Universal Robots PolyScope program: Hospital_big_top.urp

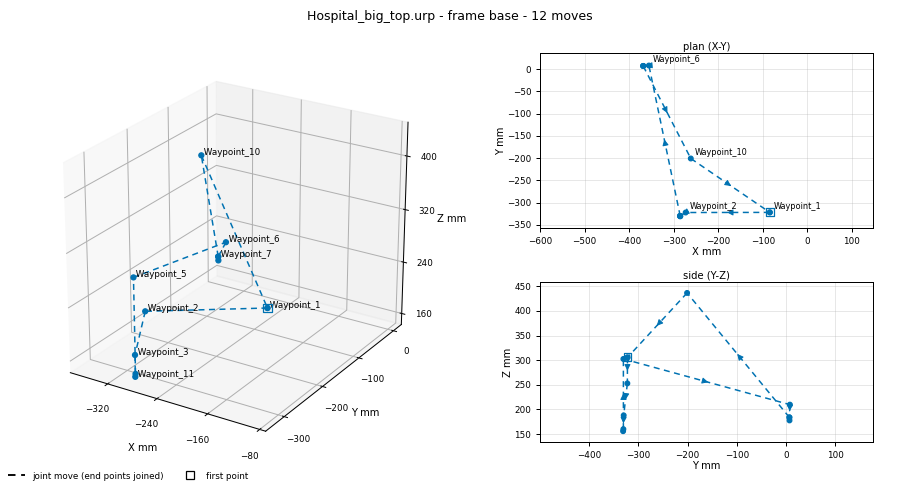
[picture p0: tool path of Hospital_big_top.urp in frame base, 12 of 12 moves have a stored position in this frame; points joined in program order, loops and branches not executed]
Program Hospital_big_top (installation=default directory=/programs/usbdisk/Zahra1 createdIn=5.11.11.1010533 lastSavedIn=5.11.11.1010533 robotSerialNumber=20205300864)
Calibrated DH parameters: a=[-0.000166, -0.243494, -0.153108, 0.000057, -0.000123, 0]; d=[0.151897, -1.34267, 53.988124, -52.514559, 0.085283, 0.092193]; alpha=[1.572472, -0.003756, 0.002824, 1.570807, -1.572621, 0]; deltaTheta=[0, 0.020704, 7.033215, -0.770746, 0.000004, 0]
Robot Program (runOnlyOnce=true)
  MoveJ speed 60 deg/s, acceleration 80 deg/s^2 (useActiveTCP=true) feature=Base
    Waypoint Waypoint_1: TCP in base x=-84.301 y=-321.874 z=305.493 mm, rx=-2.081 ry=-2.2572 rz=0.0985 rad; joints [-79.979, -91.199, -87.973, -91.694, 84.673, 815.506] deg
    URCap Gripper (Robotiq_Grippers, Robotiq Inc.) dataModel(position=46.666666666666664, force=70.0, speed=27.0, positionInDouble=46.666666666666664, forceInDouble=70.0, speedInDouble=27.0, slaveIds=[9], blocking=true, robotCompliant=false)
    Waypoint Waypoint_2: TCP in base x=-273.269 y=-322.149 z=252.836 mm, rx=-2.1606 ry=-2.2563 rz=0.1197 rad; joints [-111.769, -113.952, -75.591, -76.612, 87.489, 785.766] deg
    Waypoint Waypoint_3: TCP in base x=-286.068 y=-329.572 z=187.877 mm, rx=-2.1263 ry=-2.267 rz=0.0386 rad; joints [-113.094, -122.394, -79.226, -67.597, 87.665, 783.343] deg
    Waypoint Waypoint_11: TCP in base x=-285.496 y=-330.769 z=155.775 mm, rx=-2.2131 ry=-2.1958 rz=0.033 rad; joints [-113.09, -125.834, -82.835, -60.62, 88.212, 787.48] deg
    URCap Gripper (Robotiq_Grippers, Robotiq Inc.) dataModel(position=83.92156862745098, force=70.0, speed=27.0, positionInDouble=83.92156862745098, forceInDouble=70.0, speedInDouble=27.0, slaveIds=[9], blocking=true, robotCompliant=true)
    Waypoint Waypoint_4: motionParameters(jointSpeed=0.698132 jointAcceleration=0.523599 cartesianSpeed=0.25 cartesianAcceleration=1.2); TCP in base x=-285.424 y=-330.196 z=159.912 mm, rx=-2.2127 ry=-2.1963 rz=0.0331 rad; joints [-113.112, -125.264, -82.578, -61.439, 88.221, 787.435] deg
    Waypoint Waypoint_5: TCP in base x=-285.408 y=-330.203 z=302.436 mm, rx=-2.2127 ry=-2.1963 rz=0.0332 rad; joints [-113.041, -118.934, -53.354, -96.993, 88.181, 787.434] deg
    Waypoint Waypoint_6: TCP in base x=-355.712 y=7.819 z=209.704 mm, rx=-3.108 ry=-0.037 rz=0.0524 rad; joints [-159.113, -101.607, -103.522, -63.61, 87.579, 829.653] deg
    Waypoint Waypoint_7: TCP in base x=-368.599 y=6.796 z=183.845 mm, rx=-3.106 ry=0.0502 rz=-0.025 rad; joints [-159.969, -108.043, -101.533, -61.904, 88.456, 832.067] deg
    Waypoint Waypoint_8: motionParameters(jointSpeed=0.523599 jointAcceleration=0.349066 cartesianSpeed=0.25 cartesianAcceleration=1.2); TCP in base x=-368.491 y=7.024 z=177.653 mm, rx=-3.106 ry=0.0502 rz=-0.025 rad; joints [-160.001, -108.773, -102.426, -60.281, 88.455, 832.04] deg
    URCap Gripper (Robotiq_Grippers, Robotiq Inc.) dataModel(position=52.549019607843135, force=70.0, speed=18.0, positionInDouble=52.549019607843135, forceInDouble=70.0, speedInDouble=18.0, slaveIds=[9], blocking=true, robotCompliant=true)
    Waypoint Waypoint_7: TCP in base x=-368.599 y=6.796 z=183.845 mm, rx=-3.106 ry=0.0502 rz=-0.025 rad; joints [-159.969, -108.043, -101.533, -61.904, 88.456, 832.067] deg
    Waypoint Waypoint_10: TCP in base x=-261.732 y=-200.874 z=436.443 mm, rx=2.8911 ry=0.2915 rz=-0.1489 rad; joints [-120.045, -93.938, -55.097, -106.641, 92.936, 858.863] deg
    Waypoint Waypoint_1: TCP in base x=-84.301 y=-321.874 z=305.493 mm, rx=-2.081 ry=-2.2572 rz=0.0985 rad; joints [-79.979, -91.199, -87.973, -91.694, 84.673, 815.506] deg
